{attribute 'GeneratedUsingTerminal: EK1100-0000-0018'}
{attribute addProperty BoxType "EK1100-0000-0018"}
{attribute addProperty Id "Beckhoff_EP7xxxEK1122Beckhoff_EP7xxxEK1122_D8D4EB702992"}
{attribute addProperty CRC "1899607182"}
{attribute addProperty Size "2992"}
TYPE Beckhoff_EP7xxx_7139B48E EXTENDS EK1100_AB5A9467 :
STRUCT
	{attribute addProperty Name "Beckhoff_EP7xxxEK1122"}
	Beckhoff_EP7xxxEK1122 : Beckhoff_EP7xxxEK1122_D8D4EB70;
END_STRUCT
END_TYPE

(* stored: Version 1.2.0.0, ProductVersion 3.1.4024.9
   DUT Beckhoff_EP7xxx_7139B48E: Id {84cb71e0-31b1-408d-9618-28a0150695d7} *)
